# EPICS substitutions: devel/epics/apps/omsMotorApp/Db/omsMotor.substitutions
file "db/basic_motor.db"
{
pattern
{P,     N,  M,               DTYP,    C,  S,  DESC,          EGU,      DIR,  VELO,  VBAS,  ACCL,  BDST,  BVEL,  BACC,  MRES,  PREC,  DHLM,  DLLM,  INIT}
{HPS:,  1,  "m$(N)",  "OMS VME8/44",  0,  0,  "motor $(N)",  degrees,  Pos,  1,     .1,    .2,    0,     1,     .2,    0.01,  5,     100,   -100,  ""}
{HPS:,  2,  "m$(N)",  "OMS VME8/44",  0,  1,  "motor $(N)",  degrees,  Pos,  1,     .1,    .2,    0,     1,     .2,    0.01,  5,     100,   -100,  ""}
{HPS:,  3,  "m$(N)",  "OMS VME8/44",  0,  2,  "motor $(N)",  degrees,  Pos,  1,     .1,    .2,    0,     1,     .2,    0.01,  5,     100,   -100,  ""}
{HPS:,  4,  "m$(N)",  "OMS VME8/44",  0,  3,  "motor $(N)",  degrees,  Pos,  1,     .1,    .2,    0,     1,     .2,    0.01,  5,     100,   -100,  ""}

}
